Fanuc KAREL source: kt00327.KL

-- PROVISIONAL review KL for V770-1; original PC SHA256 4a9746ae0cb720410148f2cca6b098b7f11c3dbaf2f1be64deaf999d0ecbf5f0
-- Incomplete behavior may be omitted. Consult companion uncertainty JSON. Do not deploy.
PROGRAM KT00327
%NOLOCKGROUP
VAR
  OUT : BOOLEAN
-- UNRESOLVED_DECL V1 type=000013
-- UNRESOLVED_DECL V2 type=000013
BEGIN
  -- UNRESOLVED_PC offsets 5-20; opcodes 2E,22,32,35
  -- UNRESOLVED_PC offsets 25-40; opcodes 2E,22,32,35
  -- UNRESOLVED_PC offsets 45-60; opcodes 2E,22,32,35
  -- UNRESOLVED_PC offsets 65-80; opcodes 2E,22,32,35
  -- UNRESOLVED_PC offsets 85-108; opcodes 49,49,96,23
  -- UNRESOLVED_PC offsets 113-117; opcodes 7F
END KT00327
